///FUNCTION_BLOCK PUBLIC FB_IBuffer IMPLEMENTS IBuffer
FUNCTION_BLOCK FB_IBuffer EXTENDS FB_CtrlBase IMPLEMENTS IBuffer

// This is a Dummy-FB, used for the interface (IBuffer) to the buffer-modules

PROPERTY MaxCapacity : DINT
GET
END_GET
END_PROPERTY

PROPERTY NumOfHangers : DINT
GET
END_GET
END_PROPERTY

PROPERTY BufferFull : BOOL
GET
END_GET
END_PROPERTY

END_FUNCTION_BLOCK

(* stored: Version 1.1.0.1, ProductVersion 3.1.0.19
   POU FB_IBuffer: Id {9ec31dad-c8d1-4e2e-aa3f-873965b25876}
   Property MaxCapacity: Id {6f5294a5-4d7a-45f2-ba05-7365505de59d}
   Get Get: Id {2904cd00-dbd7-486c-9aff-892edc4b3d39}
   Property NumOfHangers: Id {170dcb0c-806c-4828-ae7a-dece73dc219a}
   Get Get: Id {3ae746a5-785b-47a4-a9b1-413913b098b1}
   Property BufferFull: Id {c94962f6-ad99-4e03-9cec-f625d834a541}
   Get Get: Id {f30b4df9-48e5-4924-9493-5c3ce8a98b07} *)
